INTERFACE PUBLIC AxisCommand EXTENDS AsyncCommand

END_INTERFACE

(* stored: Version 1.1.0.1, ProductVersion 3.1.4026.13
   Itf AxisCommand: Id {1613aa5c-36b8-0d81-2fba-98655a371f45} *)
